FUNCTION_BLOCK INTERNAL DS402_AXIS
VAR_INPUT

END_VAR
VAR_OUTPUT
	stAxisStatus : ST_AxisStatus;
END_VAR
VAR
    eModeOFOperation		: 	E_DS402_OPERATION_MODE := E_DS402_OPERATION_MODE.NONE;
	eHomingState			:	E_HOMING_STATE;
	// use this for motion time axis states
	mcAxisStates			:   MC_AxisStates;
    stPiezoAxis 			: 	REFERENCE TO  ST_PiezoStage;
END_VAR

METHOD ReadStatus
VAR_INPUT
END_VAR
IF NOT __ISVALIDREF(stPiezoAxis ) THEN
	// set an error flag
	RETURN;
END_IF
END_METHOD

PROPERTY stPiezoStageRef : REFERENCE TO ST_PiezoStage
GET
END_GET
SET
stPiezoAxis := stPiezoStageRef;
END_SET
END_PROPERTY

END_FUNCTION_BLOCK

(* stored: Version 1.1.0.1
   POU DS402_AXIS: Id {3a598b42-bac6-4032-8b4b-6a03bd2056c5}, SpecialFunc None
   Method ReadStatus: Id {26a8e682-b61c-4a6c-9633-517d6a8ce4d3}
   Property stPiezoStageRef: Id {e383f540-c0a9-403a-83d7-f686dae5e73b}
   Get Get: Id {7680a05c-d819-4478-be8f-68d9969cc170}
   Set Set: Id {d6d380d1-9fab-4bb3-a5d9-59d861fda169} *)
